FUNCTION_BLOCK ADD_DELAY (* Composite Function Block Type *)
  (* Standard: 61499-2 *)
  (* Version 0.2, 2003-12-05, JHC, Rockwell Automation, Renamed from NEWCOMPFB. *)
  (* Version 0.1, 2002-01-08, JHC, Rockwell Automation, Added DLY FB as example. *)
  (* Version 0.0, 2000-05-27, JHC, Rockwell Automation *)
  (* Compiler header: package fb.rt.template; *)
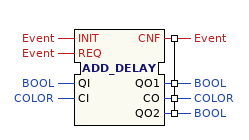
  EVENT_INPUT
    INIT;
    REQ;
  END_EVENT
  EVENT_OUTPUT
    CNF WITH QO1, CO, QO2; (* Execution Confirmation *)
  END_EVENT
  VAR_INPUT
    QI : BOOL; (* Input event qualifier *)
    CI : COLOR;
  END_VAR
  VAR_OUTPUT
    QO1 : BOOL; (* Output event qualifier *)
    CO : COLOR;
    QO2 : BOOL;
  END_VAR
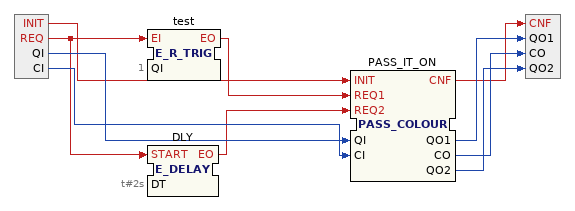
  FBS
    DLY : E_DELAY(DT := t#2s);
    test : E_R_TRIG(QI := 1);
    PASS_IT_ON : PASS_COLOUR;
  END_FBS
  EVENT_CONNECTIONS
    REQ TO test.EI;
    REQ TO DLY.START;
    INIT TO PASS_IT_ON.INIT;
    test.EO TO PASS_IT_ON.REQ1;
    DLY.EO TO PASS_IT_ON.REQ2;
    PASS_IT_ON.CNF TO CNF;
  END_CONNECTIONS
  DATA_CONNECTIONS
    QI TO PASS_IT_ON.QI;
    CI TO PASS_IT_ON.CI;
    PASS_IT_ON.QO1 TO QO1;
    PASS_IT_ON.QO2 TO QO2;
    PASS_IT_ON.CO TO CO;
  END_CONNECTIONS
END_FUNCTION_BLOCK
